TYPE
    CUComponentsBase EXTENDS TcoCore.TcoStruct :
    STRUCT
       
    END_STRUCT
END_TYPE

(* stored: Version 1.1.0.1
   DUT CUComponentsBase: Id {4b4b467f-b398-45dd-915b-88572e718a38} *)
